Omron CX-Programmer project NewProject (CX-Programmer 9.73)

# PLC NewPLC1: CP1E E30

## Global symbols (name address type ; comment)
100.01 BOOL  ; lamp
C001 BOOL  ; counter

## Program NewProgram1 (cyclic task 0)

### Section Section1

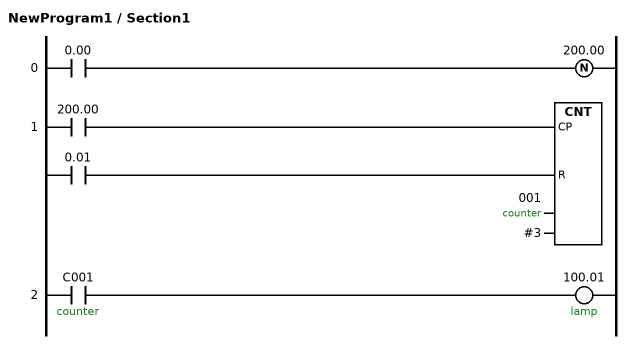
; rung 0
LD 0.00
DIFD(014) 200.00
; rung 1
LD 200.00
LD 0.01
CNT 001 #3  ; counter
; rung 2
LD C001  ; counter
OUT 100.01  ; lamp

### Section END
; rung 0
END(001)